FUNCTION_BLOCK FB_RecvDataQue
VAR_INPUT
END_VAR
VAR_OUTPUT
END_VAR
VAR
	nQueHead			: USINT := 1;
	nQueTail			: USINT := 0;
	i					: USINT := 0;
	GetDataFailCNT		: UDINT := 0;
	PutDataFailCNT		: UDINT := 0;
END_VAR
VAR (*DATA ACCESS BY SERVAL TASK*)
	bRecvQueFill		: ARRAY[1..GVL.QueLen] OF BOOL;
	bRecvQueLock		: ARRAY[1..GVL.QueLen] OF BOOL;
	RecvQue				: ARRAY[1..GVL.QueLen, 1..GVL.MaxDataLen] OF BYTE;
END_VAR

METHOD GetfromQue : BOOL
VAR_INPUT
	DataBuff 		: POINTER TO ARRAY[1..GVL.MaxDataLen] OF BYTE;
END_VAR
IF TestAndSet(bRecvQueLock[nQueHead])THEN
	IF bRecvQueFill[nQueHead] THEN
		memcpy(DataBuff,ADR(RecvQue)+ (nQueHead-1)*GVL.MaxDataLen,GVL.MaxDataLen);
		bRecvQueLock[nQueHead]:= FALSE;	
		
		bRecvQueFill[nQueHead]:= FALSE;
		nQueHead := nQueHead + 1;
		GetDataFailCNT := 0;
		IF nQueHead > 4 THEN
			nQueHead := 1;
		END_IF
	ELSE
		memset(DataBuff,0,GVL.MaxDataLen);
		bRecvQueLock[nQueHead]:= FALSE;	
		GetDataFailCNT := GetDataFailCNT+1;			
	END_IF
	
ELSE
	//the que is emty, set buffer 0.
	memset(DataBuff,0,GVL.MaxDataLen);
	GetDataFailCNT := GetDataFailCNT+1;
END_IF
END_METHOD

METHOD PUBLIC PutToQue : BOOL
VAR_INPUT
	DataBuff 		: POINTER TO ARRAY[1..GVL.MaxDataLen] OF BYTE;
END_VAR
nQueTail := nQueTail + 1;
IF nQueTail > 4 THEN
	nQueTail := 1;
END_IF
IF TestAndSet(bRecvQueLock[nQueTail])THEN
	memcpy(ADR(RecvQue)+ (nQueTail-1)*GVL.MaxDataLen,DataBuff,GVL.MaxDataLen);
	bRecvQueLock[nQueTail]:= FALSE;	
	bRecvQueFill[nQueTail]:= TRUE;
	PutDataFailCNT := 0;
	
ELSE
	//abandan this data, this may cause unresbonse to some command (very very low possiblity)
	nQueTail := nQueTail - 1;
	IF nQueTail = 0 THEN
	nQueTail := 4;
	END_IF
	PutDataFailCNT := PutDataFailCNT+1;
END_IF
END_METHOD

METHOD Reset : BOOL
VAR_INPUT
END_VAR
FOR i := 1 TO GVL.QueLen DO
	IF TestAndSet(bRecvQueLock[i]) THEN
		bRecvQueFill[i] := FALSE;
		bRecvQueLock[i] := FALSE;
	END_IF
END_FOR
nQueHead := 1;
nQueTail := 0;
END_METHOD

END_FUNCTION_BLOCK

(* stored: Version 1.1.0.1, ProductVersion 3.1.4022.12
   POU FB_RecvDataQue: Id {400763d7-e0d8-4c83-a976-4af3d2e79d18}, SpecialFunc None
   Method GetfromQue: Id {43c26d8f-6faf-4ebe-9393-459af4b4fcdd}
   Method PutToQue: Id {8eba646b-1b1f-400a-b2b7-8c3e225853f7}
   Method Reset: Id {2a0e9f08-27eb-43e7-a4e8-1a3816f0a93d} *)
